TYPE E_FeederState : (
    FEEDER_IDLE := 0,
    FEEDER_REQUEST := 10,
    FEEDER_FEEDING := 20,
    FEEDER_VERIFY := 30,
    FEEDER_COMPLETE := 40,
    FEEDER_FAULT := 100
); END_TYPE

(* stored: Version 1.1.0.1
   DUT E_FeederState: Id {E3000000-0000-4000-8000-000000000018} *)
